# EPICS autosave request: iocs/PSLdriverIOC/iocBoot/iocPSLdriver/auto_settings.req
file "PSLdriver_settings.req",    P=$(P),  R=cam1:
file "NDStdArrays_settings.req",  P=$(P),  R=image1:
file "commonPlugin_settings.req", P=$(P)
